// TIA Portal V18 export
FUNCTION "motion_level2_main" : Void   // FC22, FBD
{ S7_Optimized_Access := 'TRUE' }
VERSION : 0.1
// stored: AutoNumber true, IsIECCheckEnabled false, SetENOAutomatically false, UDAEnableTagReadback false
   VAR_TEMP
      temp_cycle_run_allowed : Bool;
      man_descrete_button1 : Bool;
      man_descrete_button2 : Bool;
      sel_v_cycle : Bool;
      sel_v_desk : Bool;
      sel_v_rem : Bool;
      place_holder : Bool;
      v_auto : Real;
      v_man : Real;
      go_request : Bool;
      loc_interrupt_semiauto_pbPlaced : Bool;
      queN : UInt;
      Cycle_MotorsGo : Bool;
      авария_расчет_циклических_позиций : Bool;
   END_VAR
BEGIN

REGION Network 2
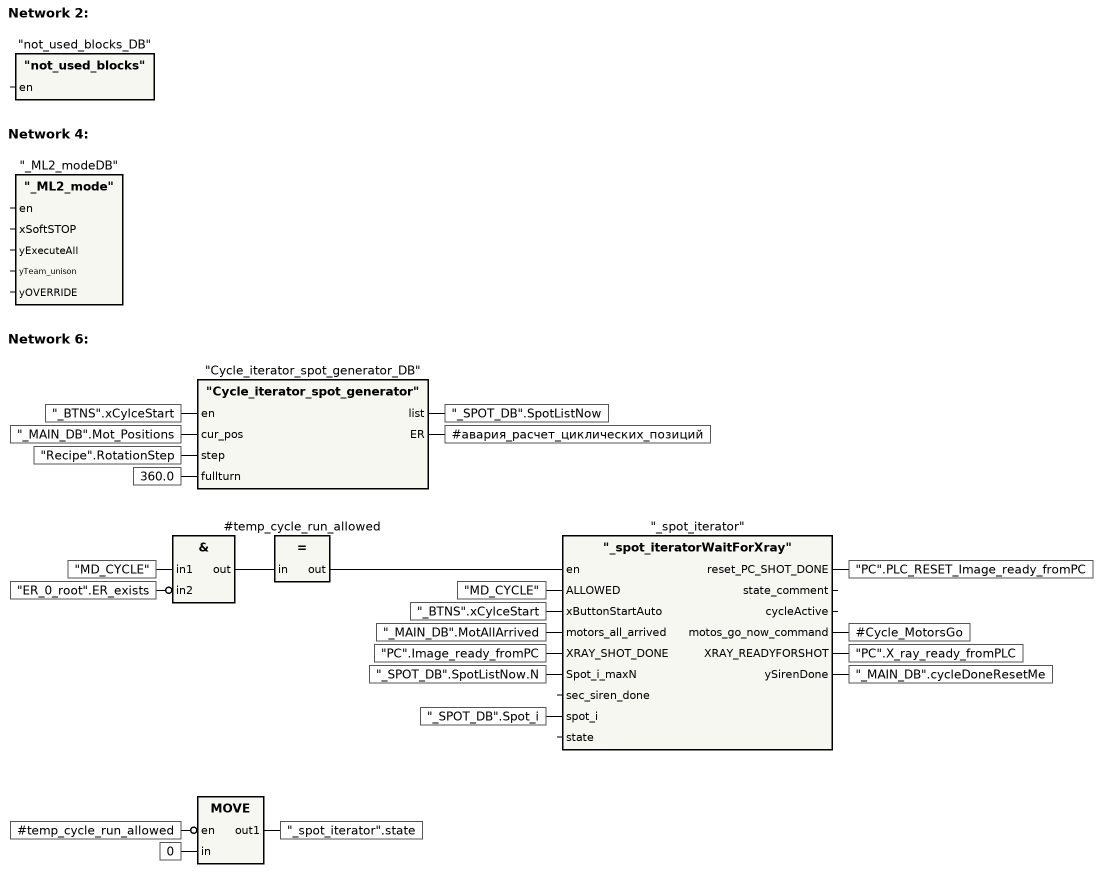
   "not_used_blocks_DB"();   // "not_used_blocks"
END_REGION

REGION Network 4
   "_ML2_modeDB"();   // "_ML2_mode"
END_REGION

REGION Network 6
   IF "_BTNS".xCylceStart THEN
       "Cycle_iterator_spot_generator_DB"(cur_pos := "_MAIN_DB".Mot_Positions,   // "Cycle_iterator_spot_generator"
                               "step" := "Recipe".RotationStep,
                               fullturn := 360.0,
                               list => "_SPOT_DB".SpotListNow,
                               ER => #авария_расчет_циклических_позиций);
   END_IF;
   #temp_cycle_run_allowed := "MD_CYCLE" AND NOT "ER_0_root".ER_exists;
   IF #temp_cycle_run_allowed THEN
       "_spot_iterator"(ALLOWED := "MD_CYCLE",   // "_spot_iteratorWaitForXray"
                        xButtonStartAuto := "_BTNS".xCylceStart,
                        motors_all_arrived := "_MAIN_DB".MotAllArrived,
                        XRAY_SHOT_DONE := "PC".Image_ready_fromPC,
                        Spot_i_maxN := "_SPOT_DB".SpotListNow.N,
                        spot_i := "_SPOT_DB".Spot_i,
                        reset_PC_SHOT_DONE => "PC".PLC_RESET_Image_ready_fromPC,
                        motos_go_now_command => #Cycle_MotorsGo,
                        XRAY_READYFORSHOT => "PC".X_ray_ready_fromPLC,
                        ySirenDone => "_MAIN_DB".cycleDoneResetMe);
   END_IF;
   IF NOT #temp_cycle_run_allowed THEN "_spot_iterator".state := 0; END_IF;
END_REGION

REGION Network 8
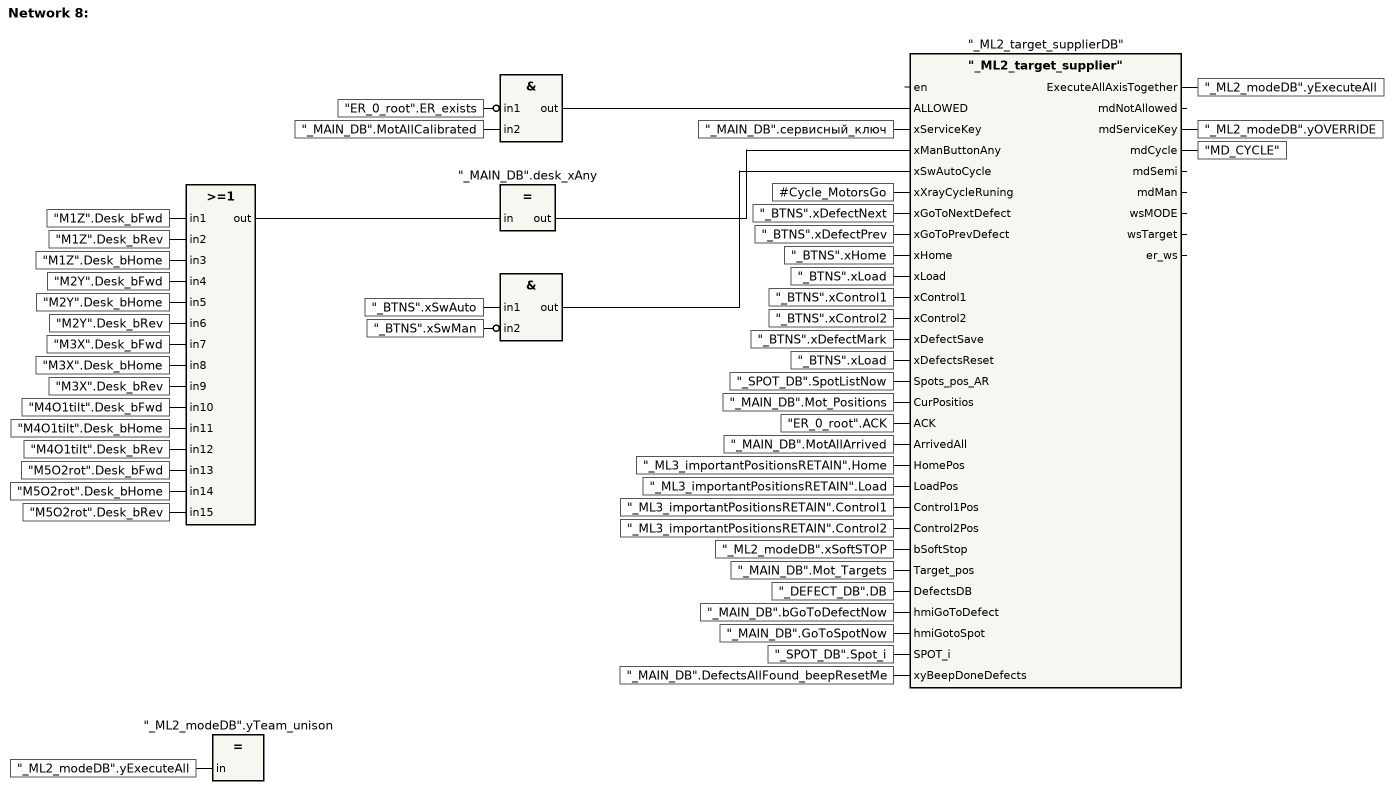
   "_MAIN_DB".desk_xAny := "M1Z".Desk_bFwd OR "M1Z".Desk_bRev OR "M1Z".Desk_bHome OR "M2Y".Desk_bFwd OR "M2Y".Desk_bHome OR "M2Y".Desk_bRev OR "M3X".Desk_bFwd OR "M3X".Desk_bHome OR "M3X".Desk_bRev OR "M4O1tilt".Desk_bFwd OR "M4O1tilt".Desk_bHome OR "M4O1tilt".Desk_bRev OR "M5O2rot".Desk_bFwd OR "M5O2rot".Desk_bHome OR "M5O2rot".Desk_bRev;
   "_ML2_target_supplierDB"(ALLOWED := NOT "ER_0_root".ER_exists AND "_MAIN_DB".MotAllCalibrated,   // "_ML2_target_supplier"
                           xServiceKey := "_MAIN_DB".сервисный_ключ,
                           xManButtonAny := "_MAIN_DB".desk_xAny,
                           xSwAutoCycle := "_BTNS".xSwAuto AND NOT "_BTNS".xSwMan,
                           xXrayCycleRuning := #Cycle_MotorsGo,
                           xGoToNextDefect := "_BTNS".xDefectNext,
                           xGoToPrevDefect := "_BTNS".xDefectPrev,
                           xHome := "_BTNS".xHome,
                           xLoad := "_BTNS".xLoad,
                           xControl1 := "_BTNS".xControl1,
                           xControl2 := "_BTNS".xControl2,
                           xDefectSave := "_BTNS".xDefectMark,
                           xDefectsReset := "_BTNS".xLoad,
                           Spots_pos_AR := "_SPOT_DB".SpotListNow,
                           CurPositios := "_MAIN_DB".Mot_Positions,
                           ACK := "ER_0_root".ACK,
                           ArrivedAll := "_MAIN_DB".MotAllArrived,
                           HomePos := "_ML3_importantPositionsRETAIN".Home,
                           LoadPos := "_ML3_importantPositionsRETAIN".Load,
                           Control1Pos := "_ML3_importantPositionsRETAIN".Control1,
                           Control2Pos := "_ML3_importantPositionsRETAIN".Control2,
                           bSoftStop := "_ML2_modeDB".xSoftSTOP,
                           Target_pos := "_MAIN_DB".Mot_Targets,
                           DefectsDB := "_DEFECT_DB".DB,
                           hmiGoToDefect := "_MAIN_DB".bGoToDefectNow,
                           hmiGotoSpot := "_MAIN_DB".GoToSpotNow,
                           SPOT_i := "_SPOT_DB".Spot_i,
                           xyBeepDoneDefects := "_MAIN_DB".DefectsAllFound_beepResetMe,
                           ExecuteAllAxisTogether => "_ML2_modeDB".yExecuteAll,
                           mdServiceKey => "_ML2_modeDB".yOVERRIDE,
                           mdCycle => "MD_CYCLE");
   "_ML2_modeDB".yTeam_unison := "_ML2_modeDB".yExecuteAll;
END_REGION

REGION Network 11
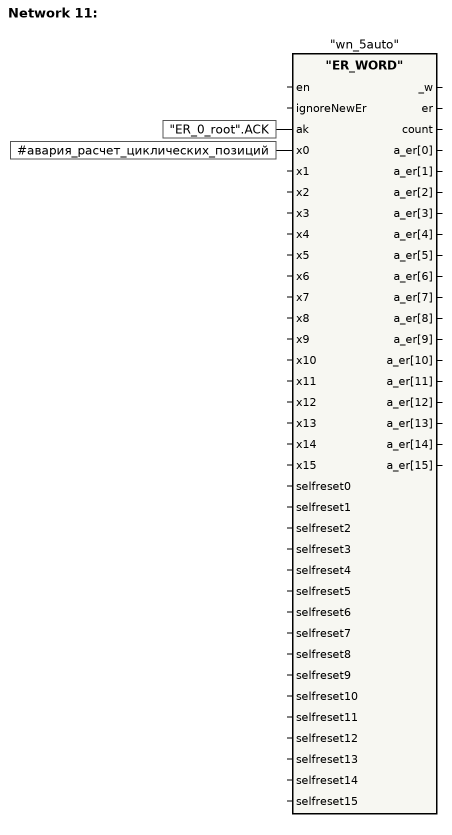
   "wn_5auto"(ak := "ER_0_root".ACK, x0 := #авария_расчет_циклических_позиций);   // "ER_WORD"
END_REGION
END_FUNCTION
